Yaskawa INFORM job: aruba_cylinder_program_with_r.JBI

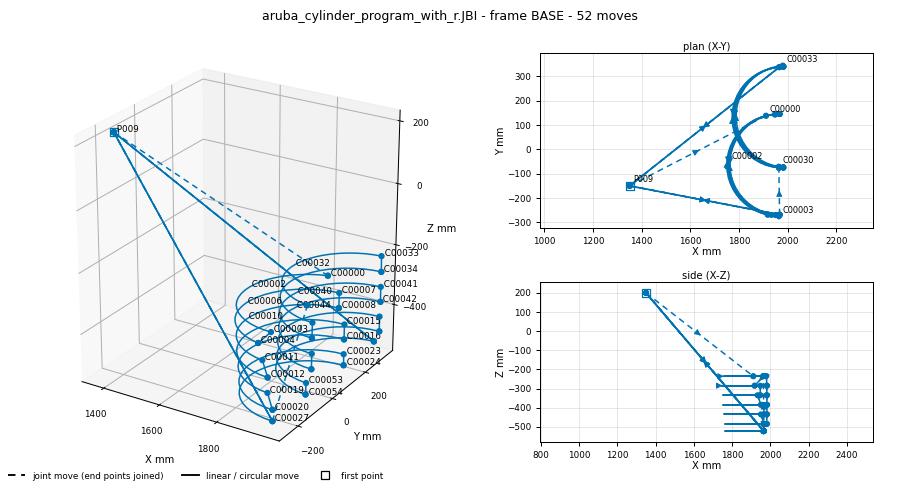
[picture p0: tool path of aruba_cylinder_program_with_r.JBI in frame BASE, 52 of 66 moves have a stored position in this frame; points joined in program order, loops and branches not executed]
/JOB
//NAME aruba_cylinder_program_with_r
//POS
///NPOS 60,0,60,1,0,1
///TOOL 0
///POSTYPE BASE
///RECTAN
///RCONF 0,0,0,0,0,0,0,0,0,0,0,0,0,0,0,0,0,0,0,0,0,0,0,0
C00000=1910.805,138.219,-235.586,90.0000,-90.0000,5.0000
C00001=1910.805,138.219,-235.586,90.0000,-90.0000,5.0000
C00002=1755.174,-55.615,-235.586,175.0000,-89.9999,5.0000
C00003=1964.123,-275.346,-235.586,-175.0000,-90.0000,90.0000
C00004=1917.868,-268.447,-284.971,-175.0000,-90.0000,90.0000
C00005=1917.868,-268.447,-284.971,-90.0000,-90.0000,5.0000
C00006=1749.583,-68.983,-284.971,175.0000,-89.9999,5.0000
C00007=1947.932,143.292,-284.971,90.0000,-90.0000,5.0000
C00008=1947.396,143.771,-334.971,90.0000,-90.0000,5.0000
C00009=1947.396,143.771,-334.971,90.0000,-90.0000,5.0000
C00010=1753.553,-69.142,-334.971,175.0000,-89.9999,5.0000
C00011=1932.885,-269.623,-334.971,-90.0000,-90.0000,5.0000
C00012=1951.055,-270.318,-384.971,-90.0000,-90.0000,5.0000
C00013=1951.055,-270.318,-384.971,-90.0000,-90.0000,5.0000
C00014=1754.528,-70.126,-384.971,175.0000,-89.9999,5.0000
C00015=1966.907,144.834,-384.971,90.0000,-90.0000,5.0000
C00016=1966.424,145.221,-434.971,90.0000,-90.0000,5.0000
C00017=1966.424,145.221,-434.971,90.0000,-90.0000,5.0000
C00018=1759.319,-51.459,-434.971,175.0000,-89.9999,5.0000
C00019=1950.333,-269.571,-434.971,-90.0000,-90.0000,5.0000
C00020=1967.203,-269.185,-484.971,-90.0000,-90.0000,5.0000
C00021=1967.203,-269.185,-484.971,-90.0000,-90.0000,5.0000
C00022=1761.552,-51.452,-484.971,175.0000,-89.9999,5.0000
C00023=1965.878,145.893,-484.971,90.0000,-90.0000,5.0000
C00024=1966.253,146.069,-522.254,90.0000,-90.0000,5.0000
C00025=1966.253,146.069,-522.254,90.0000,-90.0000,5.0000
C00026=1761.998,-52.373,-522.254,175.0000,-89.9999,5.0000
C00027=1966.773,-268.374,-522.254,-90.0000,-90.0000,5.0000
C00028=1966.773,-268.374,-522.254,-90.0000,-90.0000,5.0000
C00029=1966.773,-268.374,-522.254,-90.0000,-90.0000,5.0000
C00030=1963.415,-71.360,-234.229,-90.0000,-90.0000,5.0000
C00031=1963.415,-71.360,-234.229,-90.0000,-90.0000,5.0000
C00032=1788.149,143.986,-234.229,175.0000,-89.9999,5.0000
C00033=1979.337,344.664,-234.229,90.0000,-90.0000,5.0000
C00034=1981.794,341.634,-284.971,90.0000,-90.0000,5.0000
C00035=1981.794,341.634,-284.971,90.0000,-90.0000,5.0000
C00036=1784.524,160.319,-284.971,175.0000,-89.9999,5.0000
C00037=1982.109,-73.370,-284.971,-90.0000,-90.0000,5.0000
C00038=1981.386,-73.868,-334.971,-90.0000,-90.0000,5.0000
C00039=1981.386,-73.868,-334.971,-90.0000,-90.0000,5.0000
C00040=1783.361,161.085,-334.971,175.0000,-89.9999,5.0000
C00041=1981.823,340.854,-334.971,90.0000,-90.0000,5.0000
C00042=1982.305,340.530,-384.971,90.0000,-90.0000,5.0000
C00043=1982.305,340.530,-384.971,90.0000,-90.0000,5.0000
C00044=1781.275,161.272,-384.971,175.0000,-89.9999,5.0000
C00045=1982.037,-74.587,-384.971,-90.0000,-90.0000,5.0000
C00046=1981.965,-75.276,-434.971,-90.0000,-90.0000,5.0000
C00047=1981.965,-75.276,-434.971,-90.0000,-90.0000,5.0000
C00048=1777.143,140.664,-434.971,175.0000,-89.9999,5.0000
C00049=1981.117,339.615,-434.971,90.0000,-90.0000,5.0000
C00050=1981.953,339.092,-484.971,90.0000,-90.0000,5.0000
C00051=1981.953,339.092,-484.971,90.0000,-90.0000,5.0000
C00052=1773.316,139.287,-484.971,175.0000,-89.9999,5.0000
C00053=1964.775,-75.245,-484.971,-90.0000,-90.0000,5.0000
C00054=1963.683,-75.685,-523.153,-90.0000,-90.0000,5.0000
C00055=1963.683,-75.685,-523.153,-90.0000,-90.0000,5.0000
C00056=1771.399,123.522,-523.153,175.0000,-89.9999,5.0000
C00057=1964.923,337.768,-523.153,90.0000,-90.0000,5.0000
C00058=1964.923,337.768,-523.153,90.0000,-90.0000,5.0000
C00059=1964.923,337.768,-523.153,90.0000,-90.0000,5.0000
///POSTYPE PULSE
///PULSE
EC00000=0
EC00001=0
EC00002=0
EC00003=0
EC00004=0
EC00005=0
EC00006=0
EC00007=0
EC00008=0
EC00009=0
EC00010=0
EC00011=0
EC00012=0
EC00013=0
EC00014=0
EC00015=0
EC00016=0
EC00017=0
EC00018=0
EC00019=0
EC00020=0
EC00021=0
EC00022=0
EC00023=0
EC00024=0
EC00025=0
EC00026=0
EC00027=0
EC00028=92160
EC00029=184320
EC00030=184320
EC00031=184320
EC00032=184320
EC00033=184320
EC00034=184320
EC00035=184320
EC00036=184320
EC00037=184320
EC00038=184320
EC00039=184320
EC00040=184320
EC00041=184320
EC00042=184320
EC00043=184320
EC00044=184320
EC00045=184320
EC00046=184320
EC00047=184320
EC00048=184320
EC00049=184320
EC00050=184320
EC00051=184320
EC00052=184320
EC00053=184320
EC00054=184320
EC00055=184320
EC00056=184320
EC00057=184320
EC00058=276480
EC00059=368640
///POSTYPE BASE
///RECTAN
///RCONF 1,0,0,0,0,0,0,0,0,0,0,0,0,0,0,0,0,0,0,0,0,0,0,0
P00009=1350.000,-150.000,200.000,-180.0000,-45.0000,0.0000
///POSTYPE PULSE
///PULSE
EX00000=0
//INST
///DATE 2023/05/22 13:43
///ATTR SC,RW,RJ
////FRAME BASE
///GROUP1 RB1,ST1
NOP
MOVJ P009 EX000 VJ=15.00
MOVJ P009 VJ=15.00
MOVJ C00000 EC00000 VJ=15.00
CALL JOB:SPYON
MOVC C00001 EC00001 V=150.0
MOVC C00002 EC00002 V=150.0
MOVC C00003 EC00003 V=150.0
MOVL C00004 EC00004 V=150.0
MOVC C00005 EC00005 V=150.0
MOVC C00006 EC00006 V=150.0
MOVC C00007 EC00007 V=150.0
MOVL C00008 EC00008 V=150.0
MOVC C00009 EC00009 V=150.0
MOVC C00010 EC00010 V=150.0
MOVC C00011 EC00011 V=150.0
MOVL C00012 EC00012 V=150.0
MOVC C00013 EC00013 V=150.0
MOVC C00014 EC00014 V=150.0
MOVC C00015 EC00015 V=150.0
MOVL C00016 EC00016 V=150.0
MOVC C00017 EC00017 V=150.0
MOVC C00018 EC00018 V=150.0
MOVC C00019 EC00019 V=150.0
MOVL C00020 EC00020 V=150.0
MOVC C00021 EC00021 V=150.0
MOVC C00022 EC00022 V=150.0
MOVC C00023 EC00023 V=150.0
MOVL C00024 EC00024 V=150.0
MOVC C00025 EC00025 V=150.0
MOVC C00026 EC00026 V=150.0
MOVC C00027 EC00027 V=150.0
CALL JOB:SPYOF
MOVJ P009 VJ=15.00
MOVL C00028 EC00028 V=150.0
MOVJ P009 VJ=15.00
MOVL C00029 EC00029 V=150.0
MOVJ C00030 EC00030 VJ=15.00
CALL JOB:SPYON
MOVC C00031 EC00031 V=150.0
MOVC C00032 EC00032 V=150.0
MOVC C00033 EC00033 V=150.0
MOVL C00034 EC00034 V=150.0
MOVC C00035 EC00035 V=150.0
MOVC C00036 EC00036 V=150.0
MOVC C00037 EC00037 V=150.0
MOVL C00038 EC00038 V=150.0
MOVC C00039 EC00039 V=150.0
MOVC C00040 EC00040 V=150.0
MOVC C00041 EC00041 V=150.0
MOVL C00042 EC00042 V=150.0
MOVC C00043 EC00043 V=150.0
MOVC C00044 EC00044 V=150.0
MOVC C00045 EC00045 V=150.0
MOVL C00046 EC00046 V=150.0
MOVC C00047 EC00047 V=150.0
MOVC C00048 EC00048 V=150.0
MOVC C00049 EC00049 V=150.0
MOVL C00050 EC00050 V=150.0
MOVC C00051 EC00051 V=150.0
MOVC C00052 EC00052 V=150.0
MOVC C00053 EC00053 V=150.0
MOVL C00054 EC00054 V=150.0
MOVC C00055 EC00055 V=150.0
MOVC C00056 EC00056 V=150.0
MOVC C00057 EC00057 V=150.0
CALL JOB:SPYOF
MOVJ P009 VJ=15.00
MOVL C00058 EC00058 V=150.0
MOVJ P009 VJ=15.00
MOVL C00059 EC00059 V=150.0
END
